FUNCTION_BLOCK FB_TsFBMon_State
VAR_INPUT
	nState		: USINT;
END_VAR
VAR_OUTPUT
	sState		: STRING;
END_VAR
VAR
END_VAR

CASE nState OF
	1:		sState := 'RUN';	
	2:		sState := 'STOP';	
	3:		sState := 'SAFE';	
	4:		sState := 'ERROR';	
	5:		sState := 'RESET';	
	6:		sState := 'START';	
	7:		sState := 'ERRORDELAY';	
	8:		sState := 'DELAYOUT';	
	9:		sState := 'FUNCTEST';	
ELSE 
	sState := 'undefined';
END_CASE

END_FUNCTION_BLOCK

(* stored: Version 1.1.0.1, ProductVersion 3.1.4024.15
   POU FB_TsFBMon_State: Id {b226de47-11ca-4c30-9a16-b2cdcbe1aed9}, SpecialFunc None *)
